FUNCTION_BLOCK FB_System_BelAu
VAR_INPUT
	Freigabe_auto			: BOOL;
	Betrieb_Anford_auto		: BOOL:= TRUE;
	Regelung_Sollw_auto		: REAL;
	AdressType				: E_DALIV2AddrType;
END_VAR
VAR_OUTPUT
	{attribute 'OPC.UA.DA' := '1'}Steuerung				: ST_System_Bel_Steuerung;		
	{attribute 'OPC.UA.DA' := '1'}Stellwert				: ST_System_Bel_Stellwert;		
	{attribute 'OPC.UA.DA' := '1'}Zustand					: ST_System_Bel_Zustand;	
	{attribute 'OPC.UA.DA' := '1'}Parameter				: ST_System_Bel_Parameter;		
END_VAR
VAR
	Ablaufsteuerung			: FB_System_BelAu_Ablaufsteuerung;
	Regelung				: FB_System_BelAu_Regelung;
	Zustandscheck			: FB_System_BelAu_Zustandscheck;
	SensorikHelligkeit		: FB_System_BelAu_Sensorik;
	Logik 					: FB_System_BelAu_Logik;
	Sollwertscheck			: FB_System_BelAu_Sollwertscheck;
	Stellwertscheck			: FB_System_BelAu_Stellwertscheck;
	Regelung_Modus_auto		: SINT;


	Beleuchtung_NO: FB_Bel_RGBW;
	Beleuchtung_NW: FB_Bel_RGBW;
	Beleuchtung_SO: FB_Bel_RGBW;
	Beleuchtung_SW: FB_Bel_RGBW;
	Beleuchtung_SD: FB_Bel_RGBW;
	Beleuchtung_ND: FB_Bel_RGBW;
	Hex_Farbe	: STRING;
	Farbwert_NO: STRING;
	Farbwert_NW: STRING;
	Farbwert_ND: STRING;
	Farbwert_SO: STRING;
	Farbwert_SW: STRING;
	Farbwert_SD: STRING;


	Reset_NO: TON;
	Reset_NW: TON;
	Reset_ND: TON;
	Reset_SO: TON;
	Reset_SW: TON;
	Reset_SD: TON;
	reset: BOOL;
END_VAR

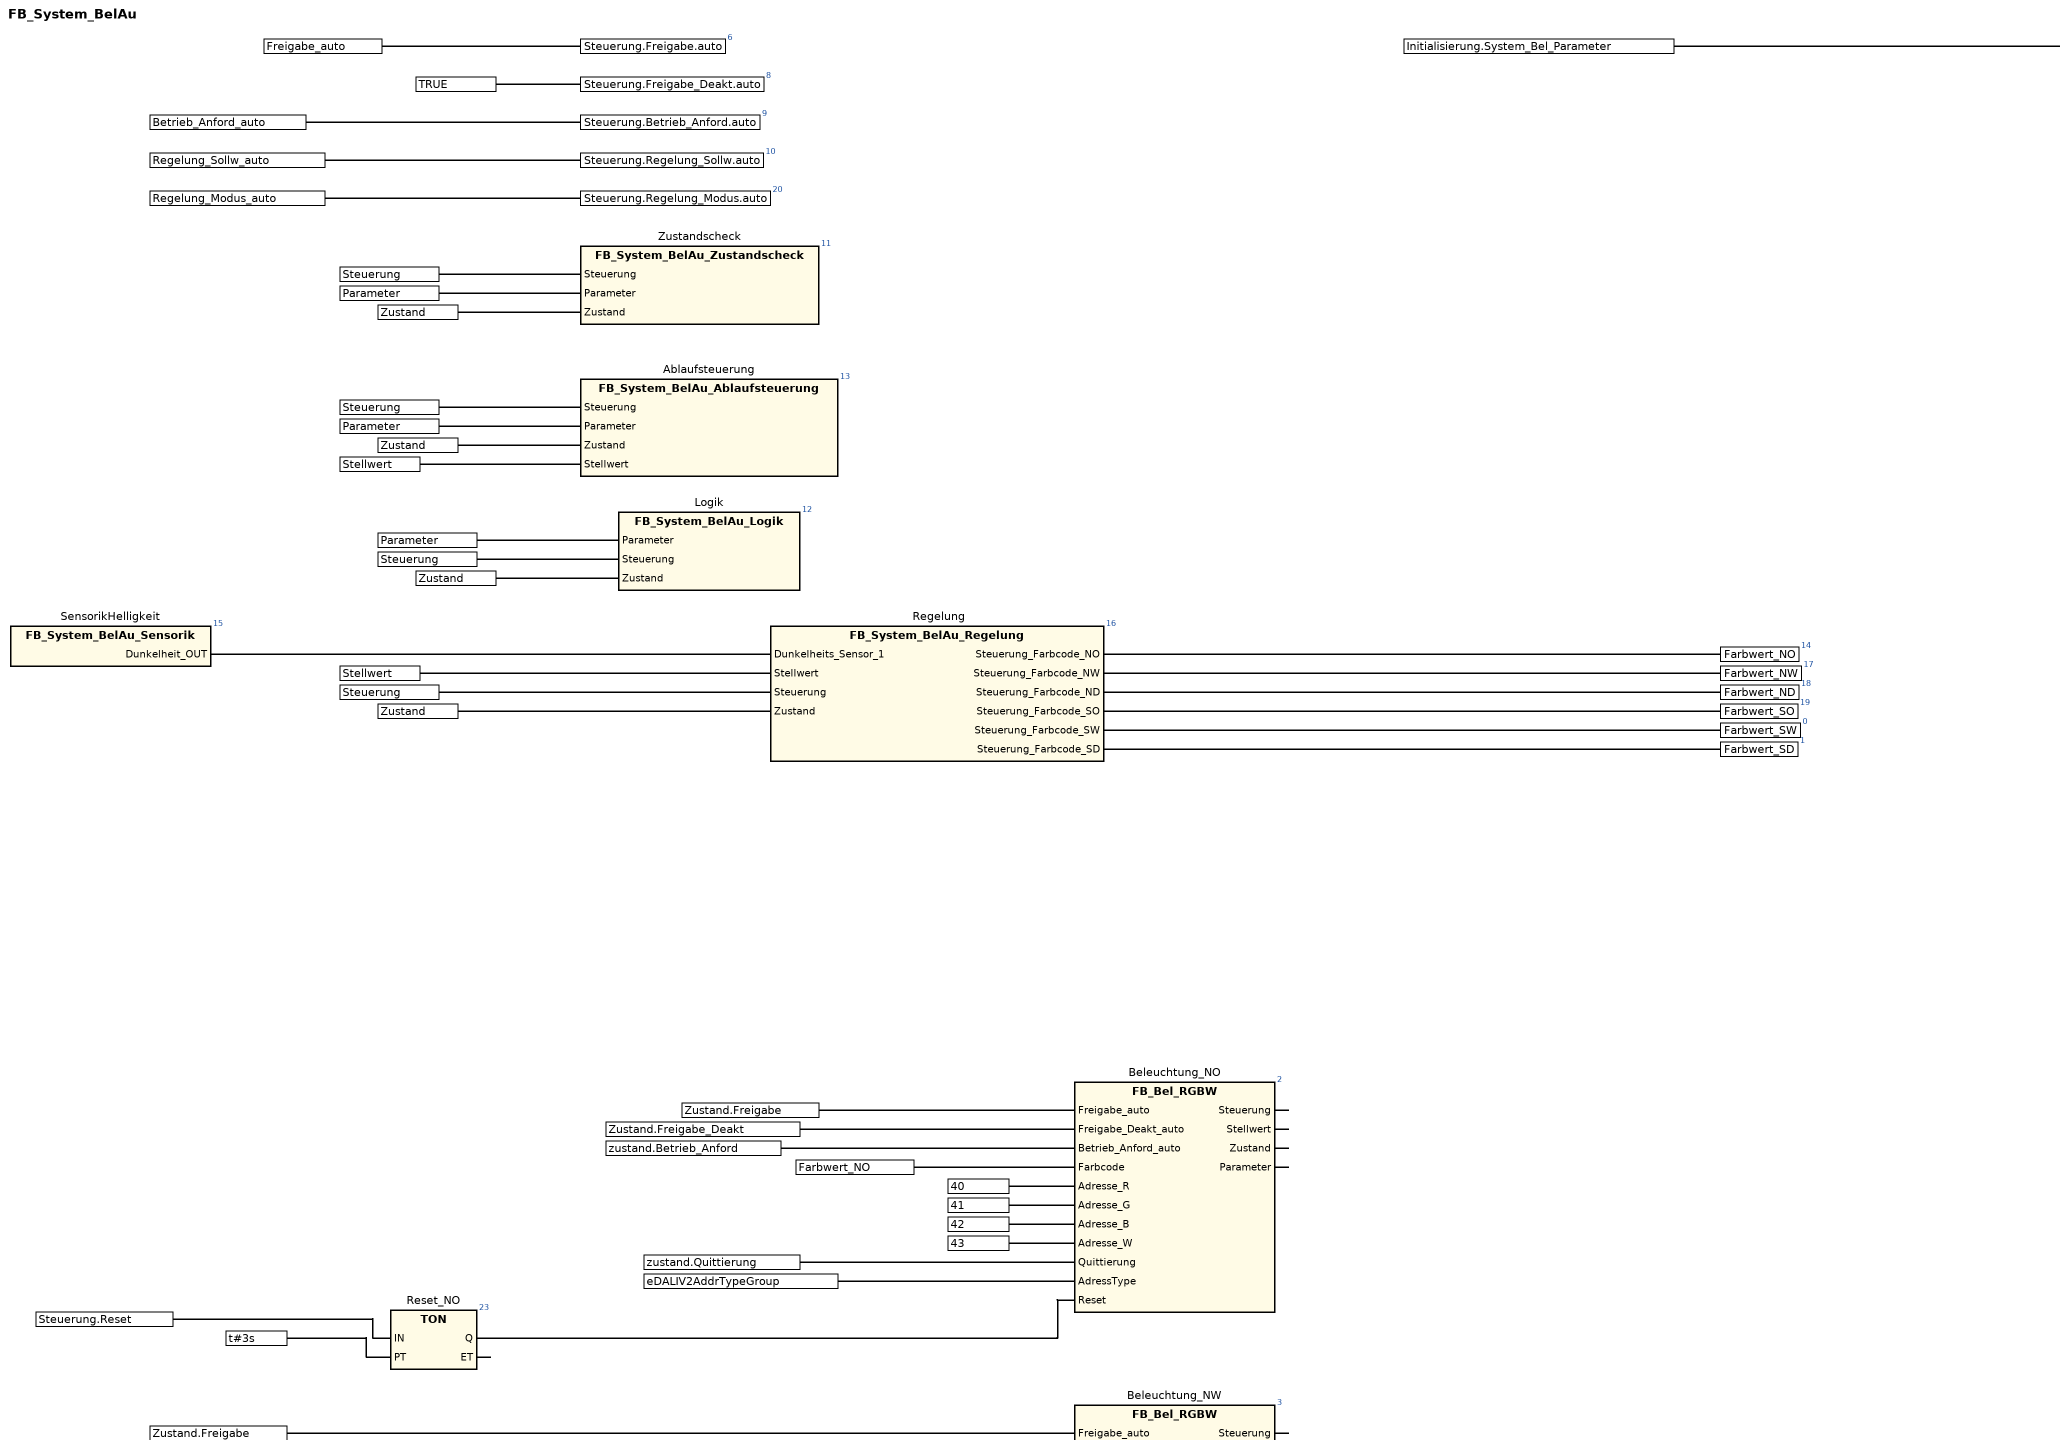
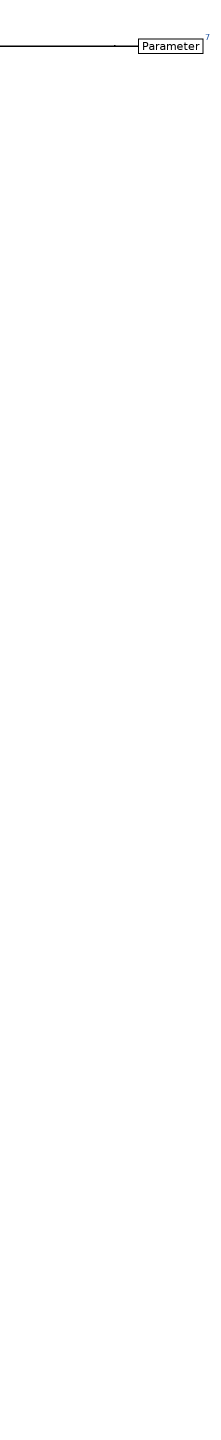
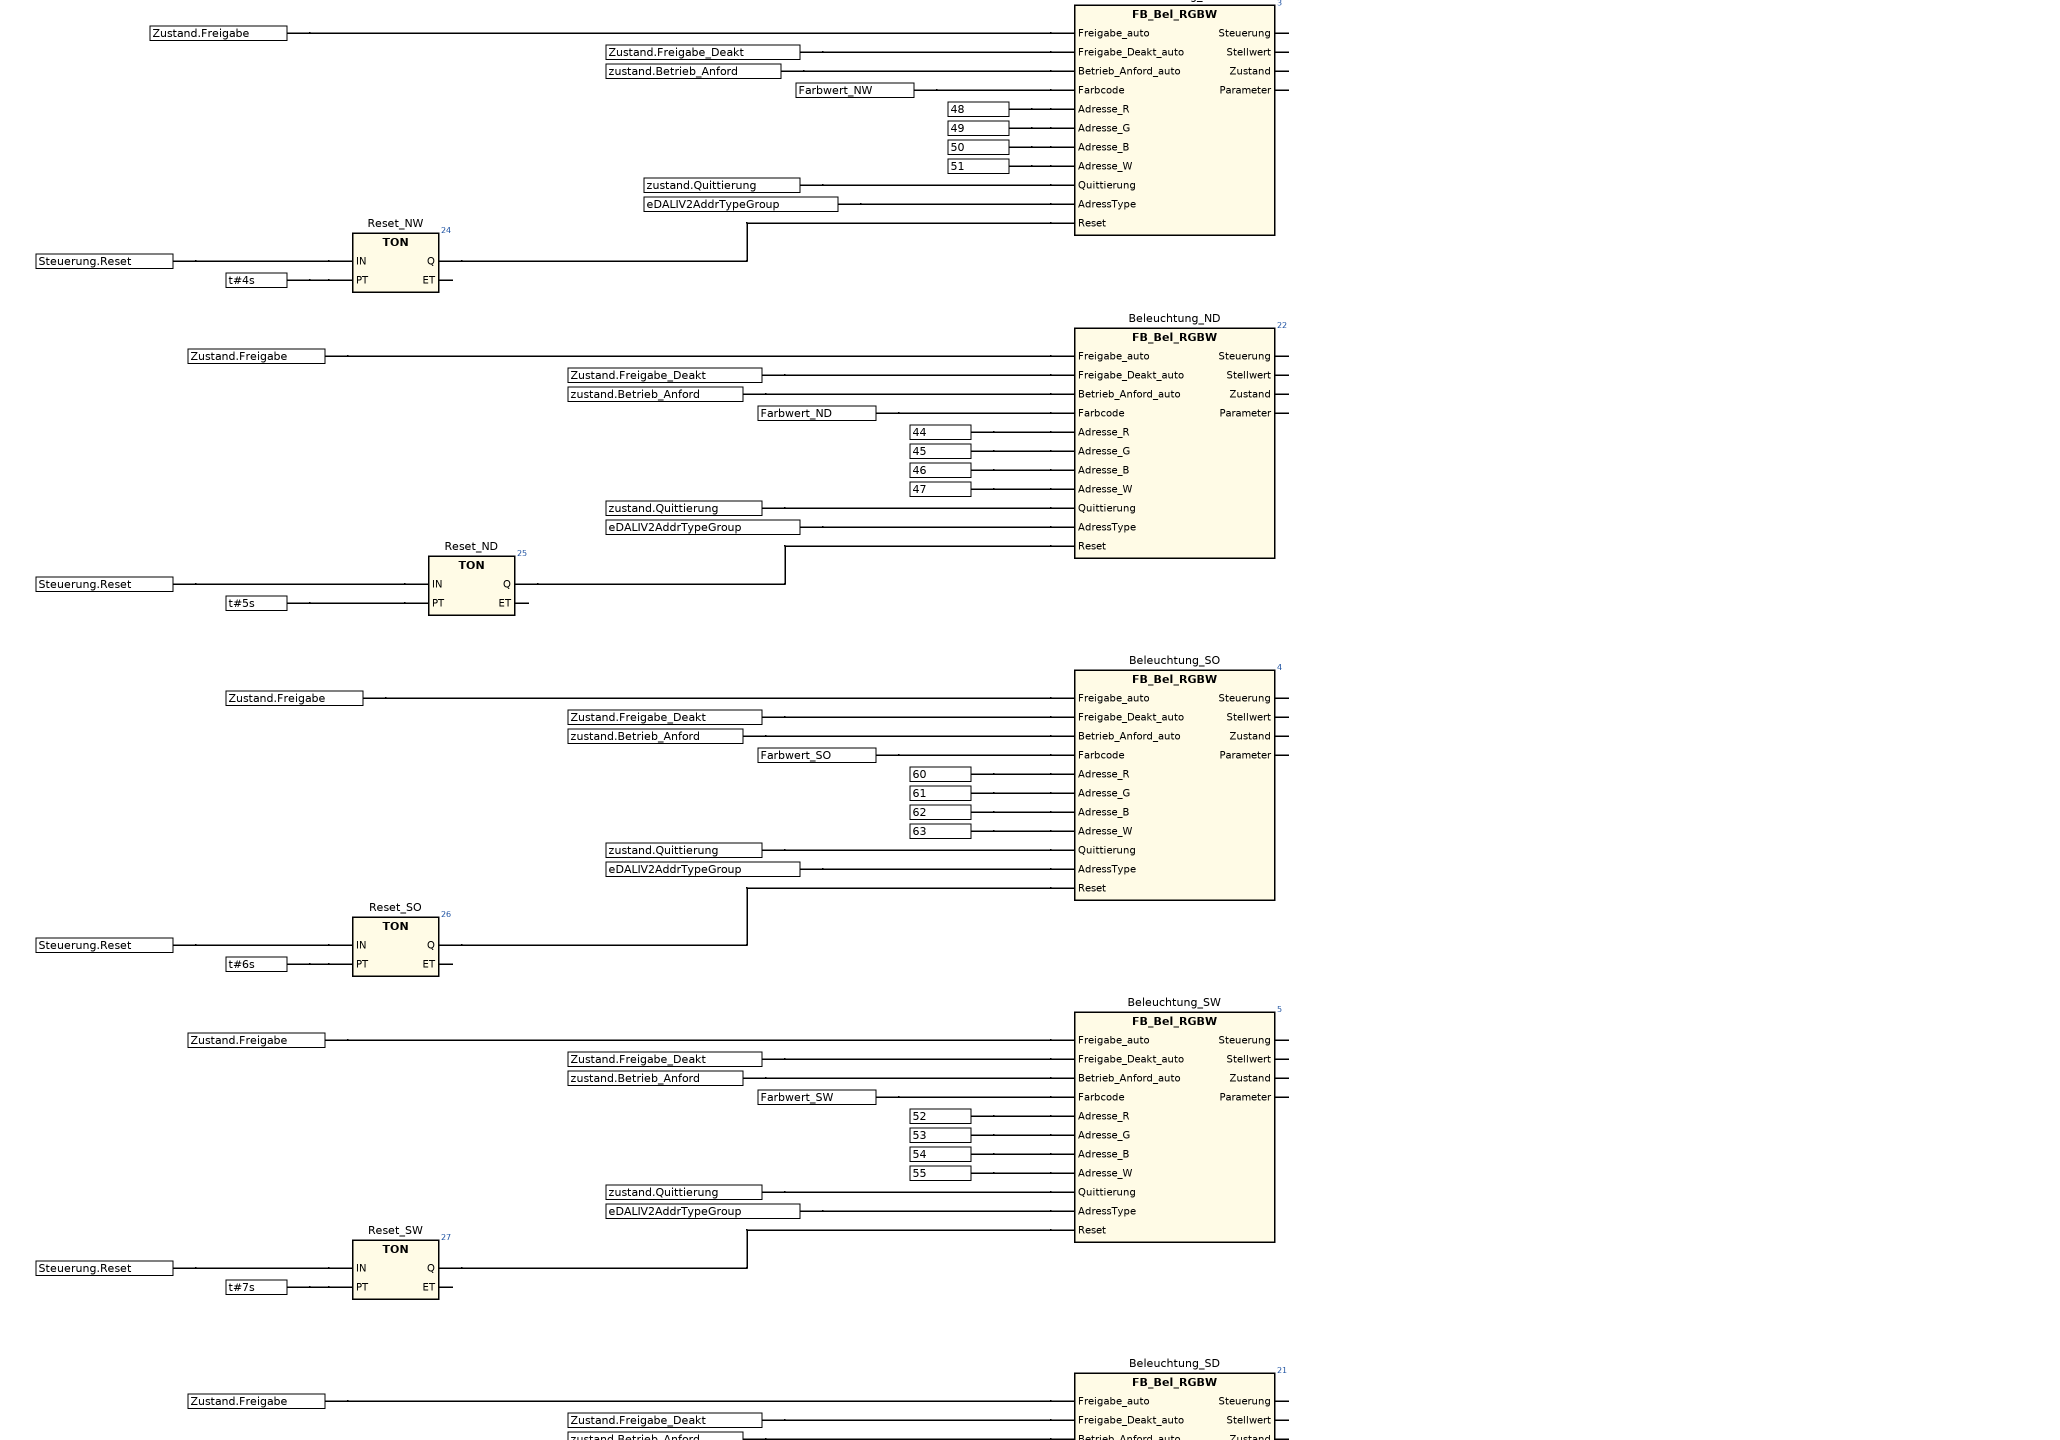
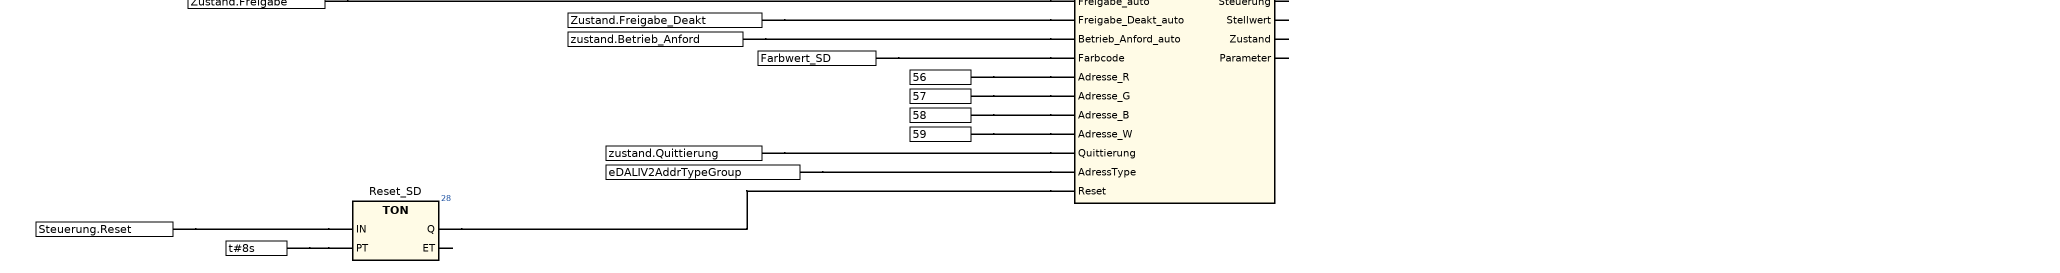
Farbwert_SW := Regelung.Steuerung_Farbcode_SW;
Farbwert_SD := Regelung.Steuerung_Farbcode_SD;
Beleuchtung_NO(
    Freigabe_auto := Zustand.Freigabe,
    Freigabe_Deakt_auto := Zustand.Freigabe_Deakt,
    Betrieb_Anford_auto := zustand.Betrieb_Anford,
    Farbcode := Farbwert_NO,
    Adresse_R := 40,
    Adresse_G := 41,
    Adresse_B := 42,
    Adresse_W := 43,
    Quittierung := zustand.Quittierung,
    AdressType := eDALIV2AddrTypeGroup,
    Reset := Reset_NO.Q); // FB_Bel_RGBW
Beleuchtung_NW(
    Freigabe_auto := Zustand.Freigabe,
    Freigabe_Deakt_auto := Zustand.Freigabe_Deakt,
    Betrieb_Anford_auto := zustand.Betrieb_Anford,
    Farbcode := Farbwert_NW,
    Adresse_R := 48,
    Adresse_G := 49,
    Adresse_B := 50,
    Adresse_W := 51,
    Quittierung := zustand.Quittierung,
    AdressType := eDALIV2AddrTypeGroup,
    Reset := Reset_NW.Q); // FB_Bel_RGBW
Beleuchtung_SO(
    Freigabe_auto := Zustand.Freigabe,
    Freigabe_Deakt_auto := Zustand.Freigabe_Deakt,
    Betrieb_Anford_auto := zustand.Betrieb_Anford,
    Farbcode := Farbwert_SO,
    Adresse_R := 60,
    Adresse_G := 61,
    Adresse_B := 62,
    Adresse_W := 63,
    Quittierung := zustand.Quittierung,
    AdressType := eDALIV2AddrTypeGroup,
    Reset := Reset_SO.Q); // FB_Bel_RGBW
Beleuchtung_SW(
    Freigabe_auto := Zustand.Freigabe,
    Freigabe_Deakt_auto := Zustand.Freigabe_Deakt,
    Betrieb_Anford_auto := zustand.Betrieb_Anford,
    Farbcode := Farbwert_SW,
    Adresse_R := 52,
    Adresse_G := 53,
    Adresse_B := 54,
    Adresse_W := 55,
    Quittierung := zustand.Quittierung,
    AdressType := eDALIV2AddrTypeGroup,
    Reset := Reset_SW.Q); // FB_Bel_RGBW
Steuerung.Freigabe.auto := Freigabe_auto;
Parameter := Initialisierung.System_Bel_Parameter;
Steuerung.Freigabe_Deakt.auto := TRUE;
Steuerung.Betrieb_Anford.auto := Betrieb_Anford_auto;
Steuerung.Regelung_Sollw.auto := Regelung_Sollw_auto;
Zustandscheck(Steuerung := Steuerung, Parameter := Parameter, Zustand := Zustand); // FB_System_BelAu_Zustandscheck
Logik(Parameter := Parameter, Steuerung := Steuerung, Zustand := Zustand); // FB_System_BelAu_Logik
Ablaufsteuerung(Steuerung := Steuerung, Parameter := Parameter, Zustand := Zustand, Stellwert := Stellwert); // FB_System_BelAu_Ablaufsteuerung
Farbwert_NO := Regelung.Steuerung_Farbcode_NO;
SensorikHelligkeit(); // FB_System_BelAu_Sensorik
Regelung(
    Dunkelheits_Sensor_1 := SensorikHelligkeit.Dunkelheit_OUT,
    Stellwert := Stellwert,
    Steuerung := Steuerung,
    Zustand := Zustand); // FB_System_BelAu_Regelung
Farbwert_NW := Regelung.Steuerung_Farbcode_NW;
Farbwert_ND := Regelung.Steuerung_Farbcode_ND;
Farbwert_SO := Regelung.Steuerung_Farbcode_SO;
Steuerung.Regelung_Modus.auto := Regelung_Modus_auto;
Beleuchtung_SD(
    Freigabe_auto := Zustand.Freigabe,
    Freigabe_Deakt_auto := Zustand.Freigabe_Deakt,
    Betrieb_Anford_auto := zustand.Betrieb_Anford,
    Farbcode := Farbwert_SD,
    Adresse_R := 56,
    Adresse_G := 57,
    Adresse_B := 58,
    Adresse_W := 59,
    Quittierung := zustand.Quittierung,
    AdressType := eDALIV2AddrTypeGroup,
    Reset := Reset_SD.Q); // FB_Bel_RGBW
Beleuchtung_ND(
    Freigabe_auto := Zustand.Freigabe,
    Freigabe_Deakt_auto := Zustand.Freigabe_Deakt,
    Betrieb_Anford_auto := zustand.Betrieb_Anford,
    Farbcode := Farbwert_ND,
    Adresse_R := 44,
    Adresse_G := 45,
    Adresse_B := 46,
    Adresse_W := 47,
    Quittierung := zustand.Quittierung,
    AdressType := eDALIV2AddrTypeGroup,
    Reset := Reset_ND.Q); // FB_Bel_RGBW
Reset_NO(IN := Steuerung.Reset, PT := t#3s); // TON
Reset_NW(IN := Steuerung.Reset, PT := t#4s); // TON
Reset_ND(IN := Steuerung.Reset, PT := t#5s); // TON
Reset_SO(IN := Steuerung.Reset, PT := t#6s); // TON
Reset_SW(IN := Steuerung.Reset, PT := t#7s); // TON
Reset_SD(IN := Steuerung.Reset, PT := t#8s); // TON

END_FUNCTION_BLOCK

(* stored: Version 1.1.0.1, ProductVersion 3.1.4024.10
   POU FB_System_BelAu: Id {0a327892-3370-436b-b47b-aef7b3995c84}, SpecialFunc None *)
